(* IEC 61131-3 sources: AccessLib/src/Ar/AccessLib, 17 files *)

(* ---- AccessLib.typ ---- *)
(*
* File: AccessLib.typ
* Copyright (c) 2023 Loupe
* https://loupe.team
*
* This file is part of AccessLib, licensed under the MIT License.
*
*)

TYPE
	UA_MODE_enum :
		(
		UA_MODE_DEFAULT,
		UA_MODE_PASSWORDONLY,
		UA_MODE_
		);
	UA_ERR_enum :
		(
		UA_ERR_SCRNBUSY := 7000,
		UA_ERR_TERMNOTCONN := 7130,
		UA_ERR_NODATA := 7195,
		UA_ERR_NULLPTR := 50000,
		UA_ERR_NUMUSERS,
		UA_ERR_NUMSTRINGS,
		UA_ERR_STRINGLENGTH,
		UA_ERR_INVALIDUSERNAME,
		UA_ERR_INVALIDPASSWORD,
		UA_ERR_USERLISTFULL,
		UA_ERR_USERNOTFOUND,
		UA_ERR_VCHANDLE,
		UA_ERR_
		);
	UA_User_typ : 	STRUCT
		UserName : STRING[UA_STRLEN_IN];
		Password : STRING[UA_STRLEN_IN];
		UserLevel : USINT;
	END_STRUCT;
END_TYPE

(* ---- UserAccessMgr.typ ---- *)
(*
* File: UserAccessMgr.typ
* Copyright (c) 2023 Loupe
* https://loupe.team
*
* This file is part of AccessLib, licensed under the MIT License.
*
*)

TYPE
	UserAccessMgr_Int_HMI_typ : 	STRUCT
		VCName : STRING[UA_STRLEN_IN];
		VCHandle : UDINT;
		AccessStatus : UINT;
		GetTouchActionStatus : UINT;
		ReleaseStatus : UINT;
		TouchAction : TouchAction;
		ScreenPress : BOOL;
		Error : BOOL;
		ErrorID : UINT;
		ErrorString : STRING[UA_STRLEN_ERROR];
	END_STRUCT;
	UserAccessMgr_Internal_typ : 	STRUCT
		LoginStatus : UDINT;
		LoginStatusTimer : TON_10ms;
		LogoutStatusTimer : TON_10ms;
		AutoLogoutTimer : TON_10ms;
		HMI : ARRAY[0..UA_MAI_VC]OF UserAccessMgr_Int_HMI_typ;
		iHMI : USINT; (*Index for stepping through configured HMIs*)
		ScreenPress : BOOL; (*Any configured screen has been pressed*)
		GTAStatus : BOOL; (*Status from UA_GetTouchAction function*)
	END_STRUCT;
	UserAccessMgr_OUT_STAT_HMI_typ : 	STRUCT
		Error : BOOL;
		ErrorID : UINT;
		ErrorString : STRING[UA_STRLEN_ERROR];
	END_STRUCT;
	UserAccessMgr_OUT_STAT_typ : 	STRUCT
		CurrentUser : UA_User_typ; (*User name and level of current user*)
		LoggerInitialized : BOOL;
		ValidLogin : BOOL;
		InvalidLogin : BOOL;
		ValidLogout : BOOL;
		AutoLogout : BOOL;
		HMI : ARRAY[0..UA_MAI_VC]OF UserAccessMgr_OUT_STAT_HMI_typ;
	END_STRUCT;
	UserAccessMgr_OUT_typ : 	STRUCT
		STAT : UserAccessMgr_OUT_STAT_typ;
	END_STRUCT;
	UserAccessMgr_IN_CFG_typ : 	STRUCT
		pUserList : UDINT; (*Pointer to the user list (address of a UA_User_typ array)*)
		NumUsers : UDINT; (*Number of users in the user list*)
		LoginMode : UDINT; (*Mode for checking login (UA_MODE_DEFAULT, UA_MODE_PASSWORDONLY)*)
		VCName : ARRAY[0..UA_MAI_VC]OF STRING[UA_STRLEN_IN]; (*Name array of the visual components objects*)
		NumVC : USINT; (*Number of VC objects to check for touch actions*)
		AutomaticLogoutDelay : UDINT; (*Automatic logout delay time [s]. Set to 0 to disable automatic logout.*)
		LoggerName : STRING[LOG_STRLEN_LOGGERNAME]; (*Name of AR logger to use*)
	END_STRUCT;
	UserAccessMgr_IN_PAR_typ : 	STRUCT
		InputUser : UA_User_typ;
	END_STRUCT;
	UserAccessMgr_IN_CMD_typ : 	STRUCT
		Login : BOOL;
		Logout : BOOL;
	END_STRUCT;
	UserAccessMgr_IN_typ : 	STRUCT
		CMD : UserAccessMgr_IN_CMD_typ;
		PAR : UserAccessMgr_IN_PAR_typ;
		CFG : UserAccessMgr_IN_CFG_typ;
	END_STRUCT;
	UserAccessMgr_typ : 	STRUCT
		IN : UserAccessMgr_IN_typ;
		OUT : UserAccessMgr_OUT_typ;
		Internal : UserAccessMgr_Internal_typ;
	END_STRUCT;
END_TYPE

(* ---- AccessLib.fun ---- *)
(*
* File: AccessLib.fun
* Copyright (c) 2023 Loupe
* https://loupe.team
*
* This file is part of AccessLib, licensed under the MIT License.
*
*)

FUNCTION UA_Logout : UDINT (*Logout function*)
	VAR_IN_OUT
		CurrentUser : UA_User_typ;
	END_VAR
END_FUNCTION

FUNCTION UA_Login : UDINT (*Login function - checks username and password*)
	VAR_INPUT
		pUserList : UDINT;
		NumUsers : UDINT;
		InputUser : UA_User_typ;
	END_VAR
	VAR_IN_OUT
		CurrentUser : UA_User_typ;
	END_VAR
	VAR
		i : UDINT;
		dUser : REFERENCE TO UA_User_typ;
	END_VAR
END_FUNCTION

FUNCTION UA_LoginPasswordOnly : UDINT (*Login function - ignores username and only checks password*)
	VAR_INPUT
		pUserList : UDINT;
		NumUsers : UDINT;
		pInputPassword : UDINT;
	END_VAR
	VAR_IN_OUT
		CurrentUser : UA_User_typ;
	END_VAR
	VAR
		i : UDINT;
		dUser : REFERENCE TO UA_User_typ;
	END_VAR
END_FUNCTION

FUNCTION UA_ListUsers : UDINT (*List all of the users with user name and level*)
	VAR_INPUT
		pUserList : UDINT;
		NumUsers : UDINT;
		pStringArray : UDINT;
		NumStrings : UDINT;
		StringLength : UDINT;
	END_VAR
	VAR
		i : UDINT;
		LoopEndIndex : UDINT;
		pCurrString : UDINT;
		UserLevelString : STRING[3];
		dUser : REFERENCE TO UA_User_typ;
	END_VAR
END_FUNCTION

FUNCTION UA_AddUser : UDINT (*Add a user to the user list*)
	VAR_INPUT
		pUserList : UDINT;
		NumUsers : UDINT;
		NewUser : UA_User_typ;
	END_VAR
	VAR
		i : UDINT;
		dUser : REFERENCE TO UA_User_typ;
	END_VAR
END_FUNCTION

FUNCTION UA_RemoveUser : UDINT (*Remove a user from the user list*)
	VAR_INPUT
		pUserList : UDINT;
		NumUsers : UDINT;
		pUserName : UDINT;
	END_VAR
	VAR
		i : UDINT;
		dUser : REFERENCE TO UA_User_typ;
	END_VAR
END_FUNCTION

FUNCTION UA_ChangePassword : UDINT (*Change a user's password*)
	VAR_INPUT
		pUserList : UDINT;
		NumUsers : UDINT;
		pUserName : UDINT;
		pOldPassword : UDINT;
		pNewPassword : UDINT;
	END_VAR
	VAR
		i : UDINT;
		dUser : REFERENCE TO UA_User_typ;
	END_VAR
END_FUNCTION

FUNCTION UA_ChangeUserLevel : UDINT (*Change a user's user level*)
	VAR_INPUT
		pUserList : UDINT;
		NumUsers : UDINT;
		pUserName : UDINT;
		NewUserLevel : USINT;
	END_VAR
	VAR
		i : UDINT;
		dUser : REFERENCE TO UA_User_typ;
	END_VAR
END_FUNCTION

FUNCTION UserAccessFn_Cyclic : BOOL (*Cyclic function for controlling user access levels*)
	VAR_IN_OUT
		t : UserAccessMgr_typ; (*User access control object*)
	END_VAR
	VAR
		i : USINT; (*Loop counter*)
		Args : BRSE_ARL_Arguments_typ; (*Logger arguments*)
	END_VAR
END_FUNCTION

FUNCTION UA_GetTouchAction : BOOL (*Wrapper for VA_GetTouchAction visapi function*)
	VAR_IN_OUT
		t : UserAccessMgr_Int_HMI_typ; (*User access internal HMI object*)
	END_VAR
END_FUNCTION

FUNCTION UA_SetHMIError : BOOL (*Set the error status on an HMI object*)
	VAR_INPUT
		ErrorID : UINT;
	END_VAR
	VAR_IN_OUT
		t : UserAccessMgr_Int_HMI_typ;
	END_VAR
END_FUNCTION

FUNCTION UA_Lock : UINT (*Lock or unlock an HMI element based on the current user level and a minimum required user level*) (*$GROUP=User*)
	VAR_INPUT
		CurrentUserLevel : USINT;
		MinUserLevel : USINT;
	END_VAR
	VAR_IN_OUT
		StatusDP : UINT;
	END_VAR
END_FUNCTION

FUNCTION UA_Hide : UINT (*Show or hide an HMI element based on the current user level and a minimum required user level*) (*$GROUP=User*)
	VAR_INPUT
		CurrentUserLevel : USINT;
		MinUserLevel : USINT;
	END_VAR
	VAR_IN_OUT
		StatusDP : UINT;
	END_VAR
END_FUNCTION

(* ---- UA_AddUser.st ---- *)
(*
* File: UA_AddUser.st
* Copyright (c) 2023 Loupe
* https://loupe.team
*
* This file is part of AccessLib, licensed under the MIT License.
*
*)

(********************************************************************)
(* Add a user to the user list										*)
(********************************************************************)

(* Checking Invalid inputs				DONE and TESTED DFB 20111020 *)
	(* pUserList						DONE and TESTED DFB 20111020 *)
	(* NumUsers							DONE and TESTED DFB 20111020 *)
	(* UserName							DONE and TESTED DFB 20111020 *)
	(* Password							DONE and TESTED DFB 20111020 *)

(* Adding user							DONE and TESTED DFB 20111020 *)
	(* Pointer math						DONE and TESTED DFB 20111020 *)
	(* memcpy							DONE and TESTED DFB 20111020 *)

(* Checking for full user list			DONE and TESTED DFB 20111020 *)

FUNCTION UA_AddUser

(********************************************************)
(* Check for invalid inputs								*)
(********************************************************)

IF( pUserList = 0 )THEN

	UA_AddUser:=	UA_ERR_NULLPTR;
	RETURN;

END_IF

IF( NumUsers = 0 )THEN

	UA_AddUser:=	UA_ERR_NUMUSERS;
	RETURN;

END_IF

IF( brsstrcmp(ADR(NewUser.UserName), ADR('')) = 0 )THEN

	UA_AddUser:=	UA_ERR_INVALIDUSERNAME;
	RETURN;

END_IF

IF( brsstrcmp(ADR(NewUser.Password), ADR('')) = 0 )THEN

	UA_AddUser:=	UA_ERR_INVALIDPASSWORD;
	RETURN;

END_IF

(********************************************************)
(* Add user to first empty user index					*)
(********************************************************)

FOR i:=0 TO (NumUsers-1) BY 1 DO

	(* Get current user *)

	dUser ACCESS pUserList + i*SIZEOF(dUser);

	(* Check for empty UserName *)

 	IF( brsstrcmp(ADR(dUser.UserName), ADR('')) = 0 )THEN

		(* Add NewUser here and exit loop *)

		brsmemcpy( ADR(dUser), ADR(NewUser), SIZEOF(NewUser) );

		UA_AddUser:=	0;
		RETURN;

 	END_IF

END_FOR

(* If you get here, then the list was full *)

UA_AddUser:=	UA_ERR_USERLISTFULL;

END_FUNCTION

(* ---- UA_ChangePassword.st ---- *)
(*
* File: UA_ChangePassword.st
* Copyright (c) 2023 Loupe
* https://loupe.team
*
* This file is part of AccessLib, licensed under the MIT License.
*
*)

(********************************************************************)
(* Change a user's password 										*)
(********************************************************************)

(* Checking Invalid inputs				DONE and TESTED DFB 20111020 *)
	(* pUserList						DONE and TESTED DFB 20111020 *)
	(* NumUsers							DONE and TESTED DFB 20111020 *)
	(* pUserName						DONE and TESTED DFB 20111020 *)
	(* pOldPassword						DONE and TESTED DFB 20111020 *)
	(* pNewPassword						DONE and TESTED DFB 20111020 *)

(* Changing password					DONE and TESTED DFB 20111020 *)
	(* Pointer math						DONE and TESTED DFB 20111020 *)
	(* Good password					DONE and TESTED DFB 20111020 *)
	(* Bad password						DONE and TESTED DFB 20111020 *)

(* User not found						DONE and TESTED DFB 20111020 *)

FUNCTION UA_ChangePassword

(********************************************************)
(* Check for invalid inputs								*)
(********************************************************)

IF( 	(pUserList = 0)
	OR	(pUserName = 0)
 	OR	(pOldPassword = 0)
 	OR	(pNewPassword = 0)
	)THEN

	UA_ChangePassword:=	UA_ERR_NULLPTR;
	RETURN;

END_IF

IF( NumUsers = 0 )THEN

	UA_ChangePassword:=	UA_ERR_NUMUSERS;
	RETURN;

END_IF

IF( brsstrcmp(pUserName, ADR('')) = 0 )THEN

	UA_ChangePassword:=	UA_ERR_INVALIDUSERNAME;
	RETURN;

END_IF

IF( 	(brsstrcmp(pOldPassword, ADR('')) = 0)
	OR	(brsstrcmp(pNewPassword, ADR('')) = 0)
 	)THEN

	UA_ChangePassword:=	UA_ERR_INVALIDPASSWORD;
	RETURN;

END_IF

(********************************************************)
(* Change password										*)
(********************************************************)

FOR i:=0 TO (NumUsers-1) BY 1 DO

	(* Get current user *)

	dUser ACCESS pUserList + i*SIZEOF(dUser);

	(* Check for matching UserName *)

 	IF( brsstrcmp(ADR(dUser.UserName), pUserName) = 0 )THEN

		(* Check for matching password *)

		IF( brsstrcmp(ADR(dUser.Password), pOldPassword) = 0 )THEN

			(* Change password and done *)

			brsstrcpy( ADR(dUser.Password), pNewPassword );

   			UA_ChangePassword:=	0;
			RETURN;

   		ELSE

			(* Passwords do not match *)

			UA_ChangePassword:=	UA_ERR_INVALIDPASSWORD;
			RETURN;

		END_IF

 	END_IF

END_FOR

(* If you get here, the user name was not found *)

UA_ChangePassword:=	UA_ERR_USERNOTFOUND;

END_FUNCTION

(* ---- UA_ChangeUserLevel.st ---- *)
(*
* File: UA_ChangeUserLevel.st
* Copyright (c) 2023 Loupe
* https://loupe.team
*
* This file is part of AccessLib, licensed under the MIT License.
*
*)

(********************************************************************)
(* Change a user's user level 										*)
(********************************************************************)

(* Checking Invalid inputs				DONE and TESTED DFB 20111021 *)
	(* pUserList						DONE and TESTED DFB 20111021 *)
	(* NumUsers							DONE and TESTED DFB 20111021 *)
	(* pUserName						DONE and TESTED DFB 20111021 *)

(* Changing user level					DONE and TESTED DFB 20111021 *)
	(* Pointer math						DONE and TESTED DFB 20111021 *)
	(* Setting user level				DONE and TESTED DFB 20111021 *)

(* User not found						DONE and TESTED DFB 20111021 *)

FUNCTION UA_ChangeUserLevel

(********************************************************)
(* Check for invalid inputs								*)
(********************************************************)

IF( 	(pUserList = 0)
	OR	(pUserName = 0)
 	)THEN

	UA_ChangeUserLevel:=	UA_ERR_NULLPTR;
	RETURN;

END_IF

IF( NumUsers = 0 )THEN

	UA_ChangeUserLevel:=	UA_ERR_NUMUSERS;
	RETURN;

END_IF

IF( brsstrcmp(pUserName, ADR('')) = 0 )THEN

	UA_ChangeUserLevel:=	UA_ERR_INVALIDUSERNAME;
	RETURN;

END_IF

(********************************************************)
(* Change user level									*)
(********************************************************)

FOR i:=0 TO (NumUsers-1) BY 1 DO

	(* Get current user *)

	dUser ACCESS pUserList + i*SIZEOF(dUser);

	(* Check for matching UserName *)

 	IF( brsstrcmp(ADR(dUser.UserName), pUserName) = 0 )THEN

		(* Change user level *)

		dUser.UserLevel:=	NewUserLevel;

		UA_ChangeUserLevel:=	0;
		RETURN;

 	END_IF

END_FOR

(* If you get here, the user name was not found *)

UA_ChangeUserLevel:=	UA_ERR_USERNOTFOUND;

END_FUNCTION

(* ---- UA_GetTouchAction.st ---- *)
(*
* File: UA_GetTouchAction.st
* Copyright (c) 2023 Loupe
* https://loupe.team
*
* This file is part of AccessLib, licensed under the MIT License.
*
*)

(********************************************************************)
(* Wrapper for VA_GetTouchAction visapi function 					*)
(********************************************************************)

(* VA_Setup							DONE and TESTED DFB 20120103 *)
	(* No error						DONE and TESTED DFB 20120103 *)
	(* Error						DONE and TESTED DFB 20120103 *)

(* VA_Saccess						DONE and TESTED DFB 20120103 *)

	(* Done							DONE and TESTED DFB 20120103 *)

		(* VA_GetTouchAction		DONE and TESTED DFB 20120103 *)
			(* Done press			DONE and TESTED DFB 20120103 *)
			(* Done no press		DONE and TESTED DFB 20120103 *)
			(* Busy					DONE will not be tested *)
			(* Error				DONE will not be tested *)

		(* VA_Srelease				DONE and TESTED DFB 20120103 *)

	(* Busy							DONE and TESTED DFB 20120103 *)

	(* Error						DONE will not be tested *)

FUNCTION UA_GetTouchAction

(* Return value is set to UA_GTA_BUSY if screen is busy and UA_GTA_FINISHED if code completed.
	This will allow you to step through VC objects based on a UA_GTA_FINISHED status from this function *)

(* Reset ScreenPress and Error info - it will be set below if appropriate *)

t.ScreenPress:=	0;

t.Error:=		0;
t.ErrorID:=		0;
t.ErrorString:=	'';

(* Get VCHandle *)

t.VCHandle:=	VA_Setup(1, t.VCName);

IF( t.VCHandle = 0 )THEN

	UA_SetHMIError( DINT_TO_UINT(UA_ERR_VCHANDLE), t );

	UA_GetTouchAction:=	UA_GTA_FINISHED;

	RETURN;

END_IF

(* Call VA_Saccess *)

t.AccessStatus:=	VA_Saccess(1, t.VCHandle);

IF( t.AccessStatus = 0 )THEN

	(* Have access to screen, try to get touch action *)

	t.GetTouchActionStatus:=	VA_GetTouchAction(1, t.VCHandle, 1, ADR(t.TouchAction) );

	(* Check GetTouchAction status *)

	IF( (t.GetTouchActionStatus = 0)	)THEN

		(* Success - someone touched the screen *)

		t.ScreenPress:=	1;

		UA_GetTouchAction:=	UA_GTA_FINISHED;

	ELSIF( (t.GetTouchActionStatus = UA_ERR_NODATA)	)THEN

		(* Success - nobody touched the screen *)

		UA_GetTouchAction:=	UA_GTA_FINISHED;

	ELSIF( (t.GetTouchActionStatus = UA_ERR_SCRNBUSY) )THEN

		(* Busy, try again *)

		UA_GetTouchAction:=	UA_GTA_BUSY;

	ELSE

		(* error with VA_GetTouchAction *)

		UA_SetHMIError( t.GetTouchActionStatus, t );

		UA_GetTouchAction:=	UA_GTA_FINISHED;

	END_IF

	(* Had access to screen, free up screen *)

	t.ReleaseStatus:=	VA_Srelease(1, t.VCHandle);

(* If there is an access error *)

ELSIF( t.AccessStatus = UA_ERR_SCRNBUSY )THEN

	(* Screen is busy, need to try again *)

	UA_GetTouchAction:=	UA_GTA_BUSY;

ELSE

	(* Other error, need to report error *)

	UA_SetHMIError( t.AccessStatus, t );

	UA_GetTouchAction:=	UA_GTA_FINISHED;

END_IF (* access error - can happen if terminal client is restarted and server is not *)

END_FUNCTION

(* ---- UA_Hide.st ---- *)
(*
* File: UA_Hide.st
* Copyright (c) 2023 Loupe
* https://loupe.team
*
* This file is part of AccessLib, licensed under the MIT License.
*
*)

(* Show or hide an HMI element based on the current user level 		*)
(* and a minimum required user level 								*)

FUNCTION UA_Hide

IF( CurrentUserLevel >= MinUserLevel )THEN
	StatusDP.0:=	0; // Visible //
ELSE
	StatusDP.0:=	1; // Hidden //
END_IF

UA_Hide:=	0;

END_FUNCTION

(* ---- UA_ListUsers.st ---- *)
(*
* File: UA_ListUsers.st
* Copyright (c) 2023 Loupe
* https://loupe.team
*
* This file is part of AccessLib, licensed under the MIT License.
*
*)

(********************************************************************)
(* List all of the users with user name and level 					*)
(********************************************************************)

(* Checking Invalid inputs				DONE and TESTED DFB 20111021 *)
	(* pUserList						DONE and TESTED DFB 20111021 *)
	(* NumUsers							DONE and TESTED DFB 20111021 *)
	(* pStringArray						DONE and TESTED DFB 20111021 *)
	(* NumStrings						DONE and TESTED DFB 20111021 *)
	(* StringLength						DONE and TESTED DFB 20111021 *)

(* Listing users						DONE and TESTED DFB 20111021 *)
	(* Pointer math						DONE and TESTED DFB 20111021 *)
	(* Rest								DONE and TESTED DFB 20111021 *)

FUNCTION UA_ListUsers

(********************************************************)
(* Check for invalid inputs								*)
(********************************************************)

IF( 	(pUserList = 0)
	OR	(pStringArray = 0)
 	)THEN

	UA_ListUsers:=	UA_ERR_NULLPTR;
	RETURN;

END_IF

IF( NumUsers = 0 )THEN

	UA_ListUsers:=	UA_ERR_NUMUSERS;
	RETURN;

END_IF

IF( NumStrings = 0 )THEN

	UA_ListUsers:=	UA_ERR_NUMSTRINGS;
	RETURN;

END_IF

IF( StringLength = 0 )THEN

	UA_ListUsers:=	UA_ERR_STRINGLENGTH;
	RETURN;

END_IF

(********************************************************)
(* List users											*)
(********************************************************)

(* Find minimum of NumUsers and NumStrings *)

IF( NumUsers < NumStrings )THEN

	LoopEndIndex:=	NumUsers - 1;

ELSE

	LoopEndIndex:=	NumStrings - 1;

END_IF

(* Clear string array *)

brsmemset( pStringArray, 0, NumStrings*StringLength );

(* List out users *)

FOR i:=0 TO LoopEndIndex BY 1 DO

	(* Get current user *)

	dUser ACCESS pUserList + i*SIZEOF(dUser);

	(* Copy UserName, then User Level *)

	pCurrString:=	pStringArray + i*StringLength;

	brsstrcpy(	pCurrString, ADR(dUser.UserName) );
	brsstrcat(	pCurrString, ADR(', Level ') );
	brsitoa(	dUser.UserLevel, ADR(UserLevelString) );
	brsstrcat(	pCurrString, ADR(UserLevelString) );

END_FOR

(* All done *)

UA_ListUsers:=	0;
RETURN;

END_FUNCTION

(* ---- UA_Lock.st ---- *)
(*
* File: UA_Lock.st
* Copyright (c) 2023 Loupe
* https://loupe.team
*
* This file is part of AccessLib, licensed under the MIT License.
*
*)

(* Lock or unlock an HMI element based on the current user level 	*)
(* and a minimum required user level 								*)

FUNCTION UA_Lock

IF( CurrentUserLevel >= MinUserLevel )THEN
	StatusDP.1:=	0; // Unlocked //
ELSE
	StatusDP.1:=	1; // Locked //
END_IF

UA_Lock:=	0;

END_FUNCTION

(* ---- UA_Login.st ---- *)
(*
* File: UA_Login.st
* Copyright (c) 2023 Loupe
* https://loupe.team
*
* This file is part of AccessLib, licensed under the MIT License.
*
*)

(********************************************************************)
(* Login function - checks UserName and Password 					*)
(********************************************************************)

(* Logout								DONE and TESTED DFB 20120103 *)

(* Checking Invalid inputs				DONE and TESTED DFB 20111021 *)
	(* pUserList						DONE and TESTED DFB 20111021 *)
	(* NumUsers							DONE and TESTED DFB 20111021 *)
	(* InputUser						DONE and TESTED DFB 20111021 *)

(* Logging in							DONE and TESTED DFB 20111021 *)
	(* Pointer math						DONE and TESTED DFB 20111021 *)
	(* Good password					DONE and TESTED DFB 20111021 *)
	(* Bad password						DONE and TESTED DFB 20111021 *)

(* User not found						DONE and TESTED DFB 20111021 *)

FUNCTION UA_Login

(********************************************************)
(* Logout												*)
(********************************************************)

UA_Logout(CurrentUser);

(********************************************************)
(* Check for invalid inputs								*)
(********************************************************)

IF (pUserList = 0) THEN
	UA_Login := UA_ERR_NULLPTR;
	RETURN;
END_IF

IF (NumUsers = 0) THEN
	UA_Login := UA_ERR_NUMUSERS;
	RETURN;
END_IF

IF (brsstrcmp(ADR(InputUser.UserName), ADR('')) = 0) THEN
	UA_Login := UA_ERR_INVALIDUSERNAME;
	RETURN;
END_IF

IF (brsstrcmp(ADR(InputUser.Password), ADR('')) = 0) THEN
	UA_Login := UA_ERR_INVALIDPASSWORD;
	RETURN;
END_IF

(********************************************************)
(* Login												*)
(********************************************************)

FOR i := 0 TO (NumUsers - 1) BY 1 DO

	(* Get current user *)

	dUser ACCESS pUserList + i * SIZEOF(dUser);

	(* Check for matching UserName *)

 	IF (brsstrcmp(ADR(dUser.UserName), ADR(InputUser.UserName)) = 0) THEN

		(* Check for matching password *)

		IF (brsstrcmp(ADR(dUser.Password), ADR(InputUser.Password)) = 0) THEN

			(* Good login *)

   			CurrentUser := dUser;
			CurrentUser.Password := '';

			UA_Login := 0;
			RETURN;

   		ELSE

			(* Passwords do not match *)

			UA_Login := UA_ERR_INVALIDPASSWORD;
			RETURN;

		END_IF

 	END_IF

END_FOR

(* If you get here, the user name was not found *)

UA_Login := UA_ERR_USERNOTFOUND;

END_FUNCTION

(* ---- UA_LoginPasswordOnly.st ---- *)
(*
* File: UA_LoginPasswordOnly.st
* Copyright (c) 2023 Loupe
* https://loupe.team
*
* This file is part of AccessLib, licensed under the MIT License.
*
*)

(********************************************************************)
(* Login function - ignores UserName and only checks Password 		*)
(********************************************************************)

(* Logout								DONE and TESTED DFB 20120103 *)

(* Checking Invalid inputs				DONE and TESTED DFB 20111021 *)
	(* pUserList						DONE and TESTED DFB 20111021 *)
	(* NumUsers							DONE and TESTED DFB 20111021 *)
	(* pInputPassword					DONE and TESTED DFB 20111021 *)

(* Logging in							DONE and TESTED DFB 20111021 *)
	(* Pointer math						DONE and TESTED DFB 20111021 *)
	(* Good password					DONE and TESTED DFB 20111021 *)
	(* Bad password						DONE and TESTED DFB 20111021 *)

FUNCTION UA_LoginPasswordOnly

(********************************************************)
(* Logout												*)
(********************************************************)

UA_Logout(CurrentUser);

(********************************************************)
(* Check for invalid inputs								*)
(********************************************************)

IF ( 	(pUserList = 0)
	OR	(pInputPassword = 0)
	) THEN

	UA_LoginPasswordOnly := UA_ERR_NULLPTR;
	RETURN;

END_IF

IF (NumUsers = 0) THEN

	UA_LoginPasswordOnly := UA_ERR_NUMUSERS;
	RETURN;

END_IF

IF (brsstrcmp(pInputPassword, ADR('')) = 0) THEN

	UA_LoginPasswordOnly := UA_ERR_INVALIDPASSWORD;
	RETURN;

END_IF

(********************************************************)
(* Login												*)
(********************************************************)

FOR i := 0 TO (NumUsers - 1) BY 1 DO

	(* Get current user *)

	dUser ACCESS pUserList + i * SIZEOF(dUser);

	(* Check for matching password *)

	IF (brsstrcmp(ADR(dUser.Password), pInputPassword) = 0) THEN

		(* Good login *)

		CurrentUser := dUser;
		CurrentUser.Password := '';

		UA_LoginPasswordOnly := 0;
		RETURN;

	END_IF

END_FOR

(* If you get here, the password was not found *)

UA_LoginPasswordOnly := UA_ERR_INVALIDPASSWORD;

END_FUNCTION

(* ---- UA_Logout.st ---- *)
(*
* File: UA_Logout.st
* Copyright (c) 2023 Loupe
* https://loupe.team
*
* This file is part of AccessLib, licensed under the MIT License.
*
*)

(********************************************************************)
(* Logout function 													*)
(********************************************************************)

(* Reset CurrentUser					DONE and TESTED DFB 20120103 *)

FUNCTION UA_Logout

	brsmemset(ADR(CurrentUser), 0, SIZEOF(CurrentUser));
	CurrentUser.UserName := UA_NOUSER;
	UA_Logout := 0;

END_FUNCTION

(* ---- UA_RemoveUser.st ---- *)
(*
* File: UA_RemoveUser.st
* Copyright (c) 2023 Loupe
* https://loupe.team
*
* This file is part of AccessLib, licensed under the MIT License.
*
*)

(********************************************************************)
(* Remove a user from the user list 								*)
(********************************************************************)

(* Checking Invalid inputs				DONE and TESTED DFB 20111020 *)
	(* pUserList						DONE and TESTED DFB 20111020 *)
	(* NumUsers							DONE and TESTED DFB 20111020 *)
	(* pUserName						DONE and TESTED DFB 20111020 *)
	(* UserName							DONE and TESTED DFB 20111020 *)

(* Removing user						DONE and TESTED DFB 20111020 *)
	(* Pointer math						DONE and TESTED DFB 20111020 *)
	(* memset							DONE and TESTED DFB 20111020 *)

(* User not found						DONE and TESTED DFB 20111020 *)

FUNCTION UA_RemoveUser

(********************************************************)
(* Check for invalid inputs								*)
(********************************************************)

IF( 	(pUserList = 0)
	OR	(pUserName = 0)
 	)THEN

	UA_RemoveUser:=	UA_ERR_NULLPTR;
	RETURN;

END_IF

IF( NumUsers = 0 )THEN

	UA_RemoveUser:=	UA_ERR_NUMUSERS;
	RETURN;

END_IF

IF( brsstrcmp(pUserName, ADR('')) = 0 )THEN

	UA_RemoveUser:=	UA_ERR_INVALIDUSERNAME;
	RETURN;

END_IF

(********************************************************)
(* Remove user 											*)
(********************************************************)

FOR i:=0 TO (NumUsers-1) BY 1 DO

	(* Get current user *)

	dUser ACCESS pUserList + i*SIZEOF(dUser);

	(* Check for matching UserName *)

 	IF( brsstrcmp(ADR(dUser.UserName), pUserName) = 0 )THEN

		(* Remove user and return *)

		brsmemset( ADR(dUser), 0, SIZEOF(dUser) );

		UA_RemoveUser:=	0;
		RETURN;

 	END_IF

END_FOR

(* If you get here, the user name was not found *)

UA_RemoveUser:=	UA_ERR_USERNOTFOUND;

END_FUNCTION

(* ---- UA_SetHMIError.st ---- *)
(*
* File: UA_SetHMIError.st
* Copyright (c) 2023 Loupe
* https://loupe.team
*
* This file is part of AccessLib, licensed under the MIT License.
*
*)

(********************************************************************)
(* Set the error status on an HMI object 							*)
(********************************************************************)

(* Set Error				DONE and TESTED DFB 20120103 *)
(* Set ErrorID				DONE and TESTED DFB 20120103 *)
(* Set ErrorString			DONE and TESTED DFB 20120103 *)

FUNCTION UA_SetHMIError

(****************************************************)
(* Set return value to get rid of compile warning 	*)
(****************************************************)

UA_SetHMIError:=	FALSE;

(************************************************)
(* Set error status								*)
(************************************************)

t.Error:=		1;
t.ErrorID:=		ErrorID;

(* Set ErrorString *)

CASE ErrorID OF

	0: t.ErrorString:=	'';

	ELSE	t.ErrorString:=	'Error accessing VC object. Automatic logout will not function. Check IN.CFG.VCName. If VC is a terminal object, check terminal connection.';

//	ELSE	t.ErrorString:=	'Unknown error.';

END_CASE

END_FUNCTION

(* ---- UserAccessFn_Cyclic.st ---- *)
(*
* File: UserAccessFn_Cyclic.st
* Copyright (c) 2023 Loupe
* https://loupe.team
*
* This file is part of AccessLib, licensed under the MIT License.
*
*)

(********************************************************************)
(* Cyclic function for controlling user access levels 				*)
(********************************************************************)

(* Login									DONE and TESTED DFB 20111021 *)
	(* Valid login							DONE and TESTED DFB 20111021 *)
	(* Invalid login						DONE and TESTED DFB 20111021 *)
	(* Status outputs						DONE and TESTED DFB 20111021 *)
	(* Logging								DONE and TESTED DFB 20140108 *)

(* Manual Logout							DONE and TESTED DFB 20120103 *)
	(* Status outputs						DONE and TESTED DFB 20120103 *)
	(* Logging								DONE and TESTED DFB 20140108 *)

(* Auto logout								DONE and TESTED DFB 20111018 *)
	(* Disabling							DONE and TESTED DFB 20111018 *)
	(* GetTouchAction handling				DONE and TESTED DFB 20120103 *)
	(* Status outputs						DONE and TESTED DFB 20111018 *)
	(* Timer handling						DONE and TESTED DFB 20110418 *)
	(* Logging out CurrentUser				DONE and TESTED DFB 20120103 *)
	(* Logging								DONE and TESTED DFB 20140108 *)

FUNCTION UserAccessFn_Cyclic

	(********************************************************************************)
	(* Set return value to get rid of compile warning 								*)
	(********************************************************************************)

	UserAccessFn_Cyclic:=	FALSE;

	IF (t.IN.CFG.LoggerName = '') THEN
		t.IN.CFG.LoggerName := UA_DEFAULT_LOGGERNAME;
	END_IF

	(********************************************************************************)
	(* Login										 								*)
	(********************************************************************************)

	IF( t.IN.CMD.Login )THEN

		(* Reset CMD *)

		t.IN.CMD.Login:=	0;

		(* Login *)

		IF( t.IN.CFG.LoginMode = UA_MODE_PASSWORDONLY )THEN

			t.Internal.LoginStatus:=	UA_LoginPasswordOnly( t.IN.CFG.pUserList,
			t.IN.CFG.NumUsers,
			ADR(t.IN.PAR.InputUser.Password),
			t.OUT.STAT.CurrentUser );

		ELSE

			t.Internal.LoginStatus:=	UA_Login( t.IN.CFG.pUserList,
			t.IN.CFG.NumUsers,
			t.IN.PAR.InputUser,
			t.OUT.STAT.CurrentUser );

		END_IF (* LoginMode *)

		IF( t.Internal.LoginStatus = 0 )THEN

			t.OUT.STAT.ValidLogin:=	1;

			Args.s[0]:=	ADR(t.OUT.STAT.CurrentUser.UserName);
			Args.i[0]:=	t.OUT.STAT.CurrentUser.UserLevel;
			logInfo( t.IN.CFG.LoggerName, 50000, 'User Login: %s, Level %i', ADR(Args) );

		ELSE

			t.OUT.STAT.InvalidLogin:=	1;

			logInfo( t.IN.CFG.LoggerName, 50000, 'Unsuccessful Login Attempt', ADR(Args) );

		END_IF

		(* Reset InputUser *)

		brsmemset( ADR(t.IN.PAR.InputUser), 0, SIZEOF(t.IN.PAR.InputUser) );

	END_IF

	(************************************************)
	(* Reset Login status after timeout				*)
	(************************************************)

	t.Internal.LoginStatusTimer.IN:=	t.OUT.STAT.ValidLogin OR t.OUT.STAT.InvalidLogin;
	t.Internal.LoginStatusTimer.PT:=	UA_STATUS_TIMEOUT * 100;

	t.Internal.LoginStatusTimer();

	IF( t.Internal.LoginStatusTimer.Q )THEN

		t.OUT.STAT.ValidLogin:=		0;
		t.OUT.STAT.InvalidLogin:=	0;

	END_IF

	(********************************************************************************)
	(* Logout										 								*)
	(********************************************************************************)

	IF( t.IN.CMD.Logout )THEN

		t.IN.CMD.Logout:=	0;

		UA_Logout( t.OUT.STAT.CurrentUser );

		t.OUT.STAT.ValidLogout:=	1;

		logInfo( t.IN.CFG.LoggerName, 50000, 'User Logout', ADR(Args) );

	END_IF

	(****************************************************************)
	(* Automatic logout												*)
	(****************************************************************)

	IF( 	(t.IN.CFG.AutomaticLogoutDelay <> 0)
		AND (t.IN.CFG.NumVC <> 0)
		AND ( t.IN.CFG.NumVC <= (UA_MAI_VC + 1) )
		)THEN

		(****************************************************************************)
		(* Step through configured number of VC objects to check for screen presses	*)
		(****************************************************************************)

		(* Check iHMI *)

		IF( t.Internal.iHMI >= t.IN.CFG.NumVC )THEN

			t.Internal.iHMI:=	0;

		END_IF

		(* Set VCName *)

		t.Internal.HMI[t.Internal.iHMI].VCName:=	t.IN.CFG.VCName[t.Internal.iHMI];

		(* GetTouchAction to set ScreenPress for each VC object *)

		t.Internal.GTAStatus:=	UA_GetTouchAction( t.Internal.HMI[t.Internal.iHMI] );

		(* If function finished, get error info and go to next HMI *)

		IF( t.Internal.GTAStatus = UA_GTA_FINISHED )THEN

			t.OUT.STAT.HMI[t.Internal.iHMI].Error:=			t.Internal.HMI[t.Internal.iHMI].Error;
			t.OUT.STAT.HMI[t.Internal.iHMI].ErrorID:=		t.Internal.HMI[t.Internal.iHMI].ErrorID;
			t.OUT.STAT.HMI[t.Internal.iHMI].ErrorString:=	t.Internal.HMI[t.Internal.iHMI].ErrorString;

			t.Internal.iHMI:=	t.Internal.iHMI + 1;

		END_IF

		(****************************************************************************)
		(* Loop through all HMIs to get ScreenPress information						*)
		(****************************************************************************)

		(* Reset ScreenPress. If any configured screens are pressed, it will be set below *)

		t.Internal.ScreenPress:=	0;

		FOR i:=0 TO t.IN.CFG.NumVC - 1 BY 1 DO

			(* Check for ScreenPress on ANY HMI *)

			t.Internal.ScreenPress:=	t.Internal.ScreenPress OR t.Internal.HMI[i].ScreenPress;

		END_FOR (* NumVC *)

		(********************************)
		(* Timer handling 				*)
		(********************************)

		t.Internal.AutoLogoutTimer.IN:=	NOT(t.Internal.ScreenPress);
		t.Internal.AutoLogoutTimer.PT:=	t.IN.CFG.AutomaticLogoutDelay * 100;

		t.Internal.AutoLogoutTimer();

		IF( t.Internal.AutoLogoutTimer.Q )THEN

			IF( 	(t.OUT.STAT.CurrentUser.UserLevel > 0)
				OR	(brsstrcmp( ADR(t.OUT.STAT.CurrentUser.UserName), ADR(UA_NOUSER) ) <> 0)
				)THEN

				UA_Logout( t.OUT.STAT.CurrentUser );

				t.OUT.STAT.AutoLogout:=	1;

				logInfo( t.IN.CFG.LoggerName, 50000, 'Automatic Logout Due To Inactivity', ADR(Args) );

			END_IF (* Logged in *)

		END_IF	(* AutoLogoutTimer.Q *)

	END_IF  (* AutoLogout configured *)

	(************************************************)
	(* Reset Logout status after timeout			*)
	(************************************************)

	t.Internal.LogoutStatusTimer.IN:=	t.OUT.STAT.ValidLogout OR t.OUT.STAT.AutoLogout;
	t.Internal.LogoutStatusTimer.PT:=	UA_STATUS_TIMEOUT * 100;

	t.Internal.LogoutStatusTimer();

	IF( t.Internal.LogoutStatusTimer.Q )THEN

		t.OUT.STAT.ValidLogout:=	0;
		t.OUT.STAT.AutoLogout:=		0;

	END_IF

END_FUNCTION

(* ---- AccessLib.var ---- *)
(*
* File: AccessLib.var
* Copyright (c) 2023 Loupe
* https://loupe.team
*
* This file is part of AccessLib, licensed under the MIT License.
*
*)
VAR CONSTANT
	UA_MAI_USER : USINT := 99;
	UA_MAI_VC : USINT := 4;
	UA_STRLEN_IN : USINT := 25;
	UA_STRLEN_ERROR : USINT := 200;
	UA_NOUSER : STRING[UA_STRLEN_IN] := 'None';
	UA_STATUS_TIMEOUT : USINT := 2; (*Time to hold Valid or Invalid Login and Logout status high [s]*)
	UA_GTA_FINISHED : BOOL := TRUE; (*UA_GetTouchAction finished*)
	UA_GTA_BUSY : BOOL := FALSE; (*UA_GetTouchAction is busy*)
	UA_DEFAULT_LOGGERNAME : STRING[LOG_STRLEN_LOGGERNAME] := 'Access';
END_VAR
